// Mitsubishi GX Works2 project: project group 16 Final   PLC: FX3G

// global labels: Global1
VAR_GLOBAL
  Start_Day AT X007 : BOOL;
  Input_Oats AT D1300 : INT;
  Input_Coco AT D8100 : INT;
  Coco AT D8110 : INT;
  Oats AT D1400 : INT;
  Input_Kadaif AT D1500 : INT;
  Kadaif AT D1600 : INT;
  Input_Pistachio AT D1700 : INT;
  Pistachio AT D1800 : INT;
END_VAR
VAR_GLOBAL CONSTANT
  Zero : INT;
END_VAR
VAR_GLOBAL
  Analog_Output AT D1900 : INT;
END_VAR
VAR_GLOBAL CONSTANT
  minimum_to_start_coco : DINT := 400;  (* E_400 *)
  minimum_to_start_oats : DINT := 100;
  minimum_to_start_kadaif : DINT;
  minimum_to_start_pistachio : DINT := 60;
END_VAR
VAR_GLOBAL
  Raw_material_empty AT M2 : BOOL;
  End_Package AT M10 : BOOL;
  Work_on AT Y007 : BOOL;
  Work_Off AT M0 : BOOL;
  Start_Casting AT X003 : BOOL;
END_VAR
VAR_GLOBAL CONSTANT
  timer_casting : INT := 4;
  four_sec : INT := 40;
END_VAR
VAR_GLOBAL
  Timer_Casting_Off AT TS13 : BOOL;
  casting AT Y002 : BOOL;
  Start_Melting AT X001 : BOOL;
  Input_Chocolate AT D1100 : INT;
  HELLP AT D8140 : INT;
  Chocolate AT D1200 : INT;
END_VAR
VAR_GLOBAL CONSTANT
  minimum_to_start_Chocolate : DINT := 400;
  sub_400g : INT := 400;
END_VAR
VAR_GLOBAL
  Termo_45 AT TC9 : BOOL;
  Trmo_45 AT X002 : BOOL;
  TS2 AT TS2 : BOOL;
  Melting_Lamp AT Y001 : BOOL;
  Melting_Indicator AT X002 : BOOL;
  Sample AT X004 : BOOL;
  Save_analog_val AT D8410 : INT;
  analog_out_1 AT D8280 : INT;
END_VAR
VAR_GLOBAL CONSTANT
  Divider : INT := 400;
END_VAR
VAR_GLOBAL
  Choice AT D7000 : REAL;
END_VAR
VAR_GLOBAL CONSTANT
  Max_Oatmix : INT := 5;
  Min_Dubai : INT := 6;
END_VAR
VAR_GLOBAL
  Oat_Lamp AT M20 : BOOL;
  Dubai_Lamp AT M30 : BOOL;
  Casting_Finish AT Y002 : BOOL;
  Casting_On AT Y002 : BOOL;
END_VAR
VAR_GLOBAL CONSTANT
  Oatmix_Oat : INT := 100;
  Oatmix_Pistachio : INT := 100;
  Dubai_Oat : INT := 20;
  Dubai_Pistachio : INT := 120;
  Dubai_Kadaif : INT := 60;
END_VAR
VAR_GLOBAL
  Cannot_mix AT M40 : BOOL;
  Can_Mix AT M40 : BOOL;
  Sec5_Component AT TC5 : BOOL;
END_VAR
VAR_GLOBAL CONSTANT
  Timer_5 : INT := 50;
  timer_5_end : INT := 5;
END_VAR
VAR_GLOBAL
  Timer_End5Sec AT TS5 : BOOL;
  Flashing_Light_1 AT TC1 : BOOL;
END_VAR
VAR_GLOBAL CONSTANT
  Flashing1 : INT := 10;
END_VAR
VAR_GLOBAL
  Flashing_Light_Finish_1 AT TS1 : BOOL;
  Flashing_Lamp_1 AT Y003 : BOOL;
  Flashing_Lamp_2 AT Y004 : BOOL;
  Flashing_Light_2 AT TC2 : BOOL;
END_VAR
VAR_GLOBAL CONSTANT
  Flashing2 : INT := 10;
END_VAR
VAR_GLOBAL
  Flashing_Light_Finish_2 AT TS2 : BOOL;
  Cooling_Switch AT X006 : BOOL;
  Lamp_For_CoolingTimer AT TC12 : BOOL;
  Cooling_Lamp AT Y006 : BOOL;
  Packaging_Swich AT X000 : BOOL;
  Packaging_On AT Y005 : BOOL;
  Package_Counter AT CC3 : BOOL;
END_VAR
VAR_GLOBAL CONSTANT
  Packaging_3 : INT := 3;
END_VAR
VAR_GLOBAL
  Packaging_Counter AT CC3 : BOOL;
  Finish_Count_Packaging AT M15 : BOOL;
  Count_Packaging AT M15 : BOOL;
  Packaging_Finish AT CS3 : BOOL;
  Count_Fainal_Chocolate_Pack AT D2000 : REAL;
END_VAR
VAR_GLOBAL CONSTANT
  Constanat : INT := 1;
  Add_Pack : INT := 1;
  minimum_to_start_pistachio_100 : INT := 100;
  minimum_to_start_Chocolate_400 : INT := 400;
  minimum_to_start_oats_100 : INT := 100;
END_VAR
VAR_GLOBAL
  Material_Empty AT M2 : BOOL;
END_VAR
VAR_GLOBAL CONSTANT
  Termo_450 : INT := 450;
END_VAR
VAR_GLOBAL
  Tmer_Casting_Off AT TS1 : BOOL;
  Casting_Lamp AT M8 : BOOL;
  Pan_Count AT CC7 : BOOL;
END_VAR
VAR_GLOBAL CONSTANT
  Pan_Max : INT := 4;
END_VAR
VAR_GLOBAL
  Pan_Count_4 AT CS7 : BOOL;
  Finish_Count_Pan AT TC13 : BOOL;
  Placement_Timer AT TC8 : BOOL;
END_VAR
VAR_GLOBAL CONSTANT
  max_to_start_Chocolate_400 : INT := 400;
  minmum_to_start_oats_100 : INT := 100;
  min_to_start_Chocolate_400 : INT := 400;
  min_to_start_oats_100 : INT := 100;
  min_to_start_pistachio_100 : INT := 100;
  min_to_start_kadaif : DINT := 60;
  min_to_start_kadaif_60 : INT := 60;
END_VAR
VAR_GLOBAL
  Transfer_Coco_Lamp AT Y010 : BOOL;
END_VAR
VAR_GLOBAL CONSTANT
  Chocolate_In : INT := 400;
END_VAR
VAR_GLOBAL
  Melting_Bowl AT D2000 : INT;
END_VAR
VAR_GLOBAL CONSTANT
  Chocolate_400g : INT := 400;
END_VAR
VAR_GLOBAL
  Analog_In_1 AT D8280 : INT;
END_VAR
VAR_GLOBAL CONSTANT
  Max_Oatmix_5 : INT := 5;
  Divider_400 : INT := 400;
  Min_Dubai_6 : INT := 6;
  Min_Dubai_5 : REAL := 5;
END_VAR
VAR_GLOBAL
  Nuts AT D1400 : INT;
  Input_Nuts AT D1300 : INT;
END_VAR
VAR_GLOBAL CONSTANT
  min_to_start_nuts_100 : INT := 100;
  Max_Nuts_5 : INT := 5;
  Nutsmix_Nuts : INT := 100;
  Max_Nutsmix_5 : REAL := 5;
  Dubai_Nuts : INT := 20;
  Nuts_Mixing_Cream_200 : INT := 200;
END_VAR
VAR_GLOBAL
  Mixing_Bowl AT D2100 : INT;
END_VAR
VAR_GLOBAL CONSTANT
  Dubai_Cream_155 : INT := 155;
  Nuts_Cream_200 : INT := 200;
END_VAR
VAR_GLOBAL
  Lamp_Nuts AT M52 : BOOL;
END_VAR
VAR_GLOBAL CONSTANT
  Timer_3 : INT := 30;
END_VAR
VAR_GLOBAL
  Tempature_Reached AT X002 : BOOL;
  Melting_Indicaor_Ending AT M16 : BOOL;
  Melting_Indicator_Ending AT M16 : BOOL;
  Pan_Indicator AT X003 : BOOL;
  Pan_Located AT M45 : BOOL;
  Emergency_Swich AT X005 : BOOL;
END_VAR
VAR_GLOBAL CONSTANT
  Packaging_4 : INT := 4;
END_VAR
VAR_GLOBAL
  Timer_Cast AT TC18 : BOOL;
  Casting_Timer_4 AT TC11 : BOOL;
  Finish_Casting_Timer AT TS11 : BOOL;
  Lamp_For_CoolingTimer_Finish AT TS12 : BOOL;
  End_Of_Round AT M35 : BOOL;
  Finished_Cream AT M42 : BOOL;
END_VAR
VAR_GLOBAL CONSTANT
  Divider_10 : INT := 10;
END_VAR
VAR_GLOBAL
  AANALOG_OUTPUT AT D8282 : INT;
END_VAR
VAR_GLOBAL CONSTANT
  Multiply_40 : INT := 40;
END_VAR
VAR_GLOBAL
  storage_info AT D3020 : INT;
END_VAR
VAR_GLOBAL CONSTANT
  Multiply_400 : INT := 400;
  min_to_start_pistachio_120 : INT := 120;
  Nutmix_Pistachio : INT := 100;
END_VAR
VAR_GLOBAL
  Timer_End_5_Sec AT TS5 : BOOL;
  Sec_5_Component AT TC5 : BOOL;
  Emergency_Switch AT X005 : BOOL;
  Lamp_Cooling_Timer AT TC12 : BOOL;
  Lamp_Cooling_Timer_Finish AT TS12 : BOOL;
  Packaging_Switch AT X000 : BOOL;
  Aanalog_Output_2 AT D8282 : INT;
END_VAR

// task Task_01 (event TRUE, interval 0, priority 31): POU_01

PROGRAM POU_01
VAR CONSTANT
  Nuts_Lamp : BOOL;
END_VAR
VAR
  Timer_Casting_4 : BOOL;
  Finish_Cream : BOOL;
END_VAR
(* structured ladder/FBD written out as ST: instructions are called as NAME(EN, inputs, outputs); _pN, _eN, _tN stand for wires *)
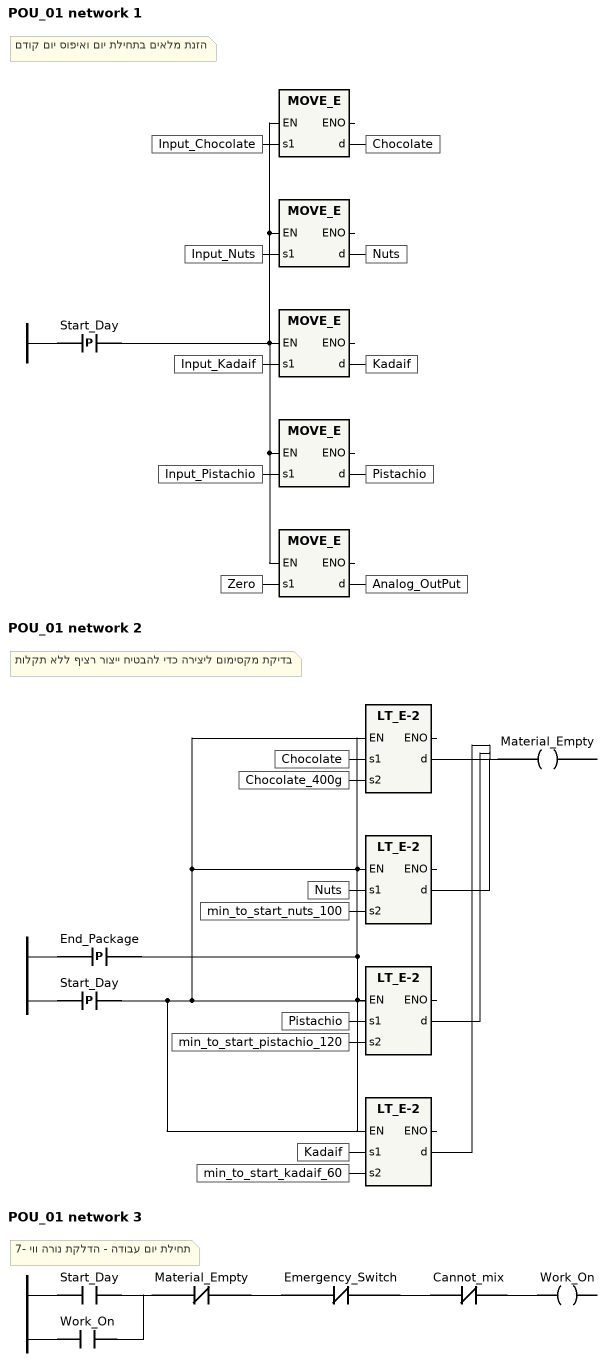
(* network 1 *)
(* הזנת מלאים בתחילת יום ואיפוס יום קודם *)
_p1 := LDP(TRUE, Start_Day);
MOVE_E(_p1, Input_Chocolate, Chocolate);
MOVE_E(_p1, Input_Nuts, Nuts);
MOVE_E(_p1, Input_Kadaif, Kadaif);
MOVE_E(_p1, Input_Pistachio, Pistachio);
MOVE_E(_p1, Zero, Analog_OutPut);
(* network 2 *)
(* בדיקת מקסימום ליצירה כדי להבטיח ייצור רציף ללא תקלות *)
_p1 := LDP(TRUE, End_Package) OR LDP(TRUE, Start_Day);
LT_E(_p1, Chocolate, Chocolate_400g, _t2);
LT_E(_p1, Nuts, min_to_start_nuts_100, _t3);
LT_E(_p1, Pistachio, min_to_start_pistachio_120, _t4);
LT_E(_p1, Kadaif, min_to_start_kadaif_60, _t5);
Material_Empty := _t2 OR _t3 OR _t4 OR _t5;
(* network 3 *)
(* תחילת יום עבודה - הדלקת נורה ווי -7 *)
Work_On := (((Start_Day OR Work_On) AND NOT Material_Empty) AND NOT Emergency_Switch) AND NOT Cannot_mix;
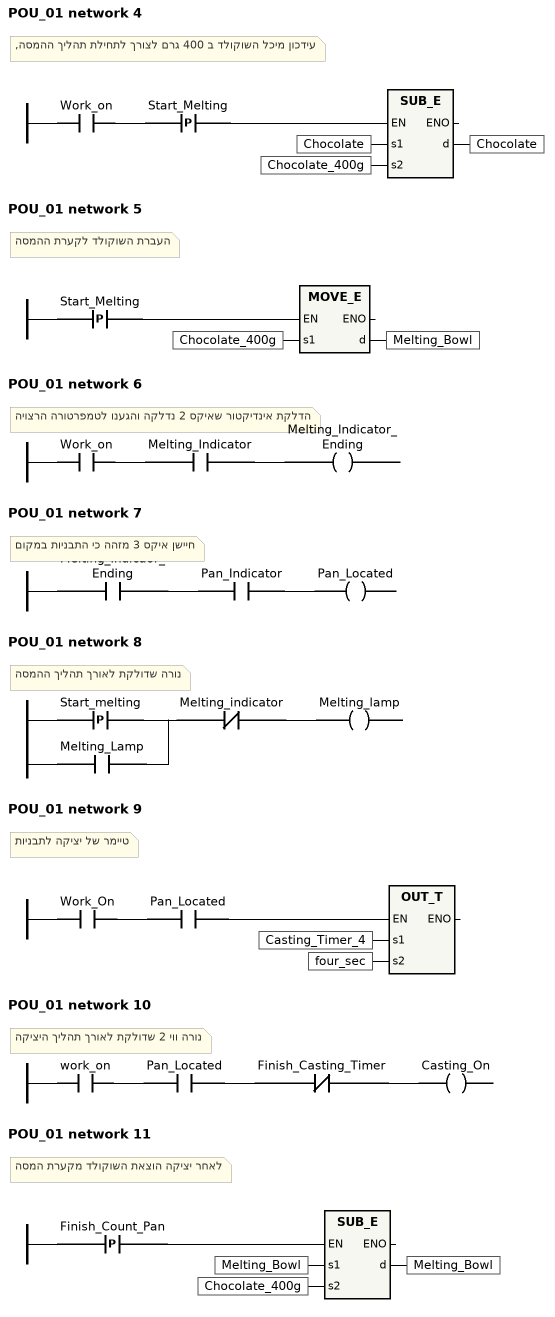
(* network 4 *)
(* עידכון מיכל השוקולד ב 400 גרם לצורך לתחילת תהליך ההמסה, *)
SUB_E(Work_on AND LDP(TRUE, Start_Melting), Chocolate, Chocolate_400g, Chocolate);
(* network 5 *)
(* העברת השוקולד לקערת ההמסה *)
MOVE_E(LDP(TRUE, Start_Melting), Chocolate_400g, Melting_Bowl);
(* network 6 *)
(* הדלקת אינדיקטור שאיקס 2 נדלקה והגענו לטמפרטורה הרצויה *)
Melting_Indicator_Ending := Work_on AND Melting_Indicator;
(* network 7 *)
(* חיישן איקס 3 מזהה כי התבניות במקום *)
Pan_Located := Melting_Indicaor_Ending AND Pan_Indicator;
(* network 8 *)
(* נורה שדולקת לאורך תהליך ההמסה *)
Melting_lamp := (LDP(TRUE, Start_melting) OR Melting_Lamp) AND NOT Melting_indicator;
(* network 9 *)
(* טיימר של יציקה לתבניות *)
OUT_T(Work_On AND Pan_Located, Casting_Timer_4, four_sec);
(* network 10 *)
(* נורה ווי 2 שדולקת לאורך תהליך היציקה *)
Casting_On := work_on AND Pan_Located AND NOT Finish_Casting_Timer;
(* network 11 *)
(* לאחר יציקה הוצאת השוקולד מקערת המסה *)
SUB_E(LDP(TRUE, Finish_Count_Pan), Melting_Bowl, Chocolate_400g, Melting_Bowl);
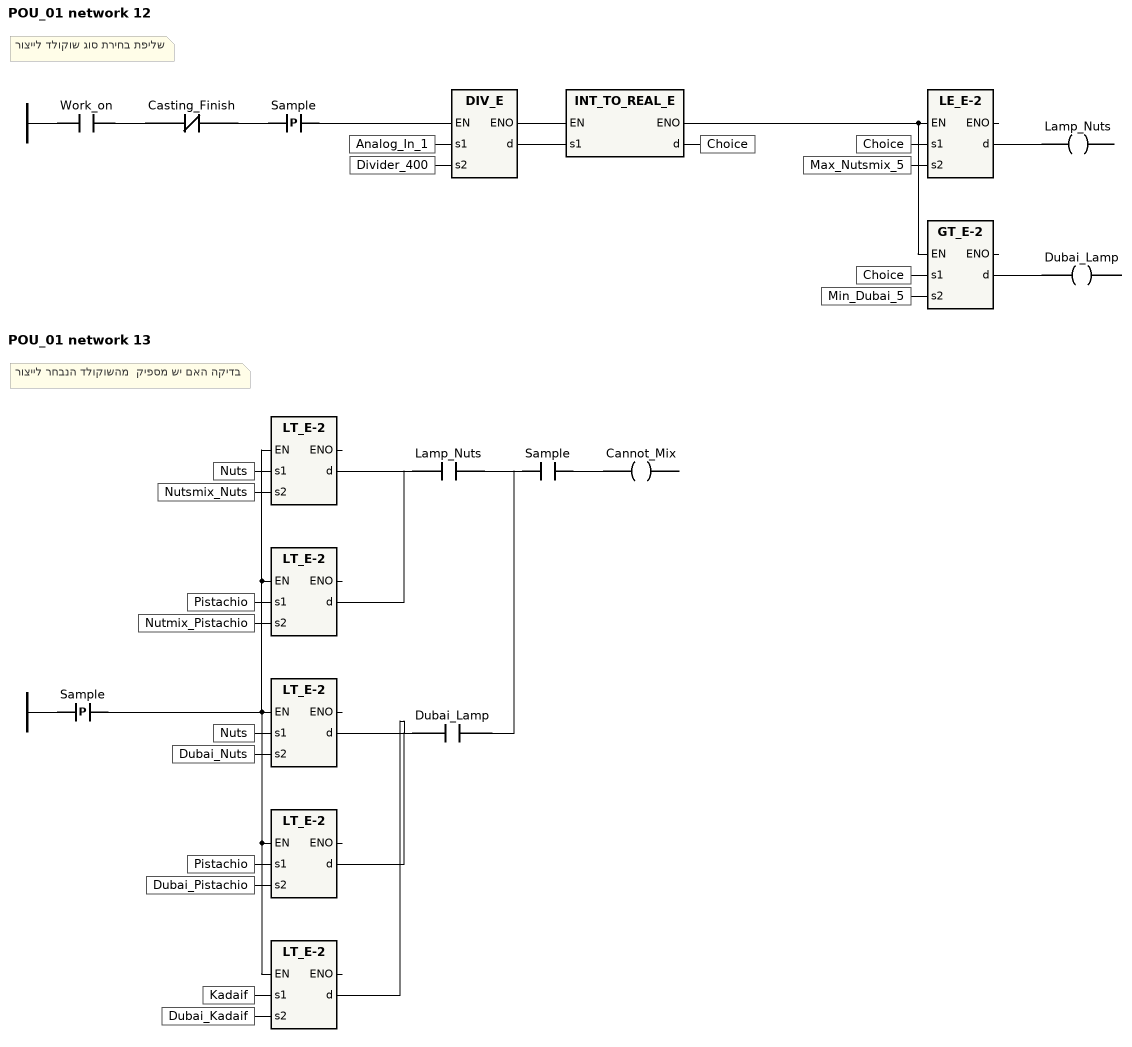
(* network 12 *)
(* שליפת בחירת סוג שוקולד לייצור *)
_e2 := DIV_E(Work_on AND NOT Casting_Finish AND LDP(TRUE, Sample), Analog_In_1, Divider_400, _t1);
_e3 := INT_TO_REAL_E(_e2, _t1, Choice);
LE_E(_e3, Choice, Max_Nutsmix_5, _t4);
Lamp_Nuts := _t4;
GT_E(_e3, Choice, Min_Dubai_5, _t5);
Dubai_Lamp := _t5;
(* network 13 *)
(* בדיקה האם יש מספיק  מהשוקולד הנבחר לייצור *)
_p1 := LDP(TRUE, Sample);
LT_E(_p1, Nuts, Nutsmix_Nuts, _t2);
LT_E(_p1, Pistachio, Nutmix_Pistachio, _t3);
LT_E(_p1, Nuts, Dubai_Nuts, _t4);
LT_E(_p1, Pistachio, Dubai_Pistachio, _t5);
LT_E(_p1, Kadaif, Dubai_Kadaif, _t6);
Cannot_Mix := (((_t2 OR _t3) AND Lamp_Nuts) OR ((_t4 OR _t5 OR _t6) AND Dubai_Lamp)) AND Sample;
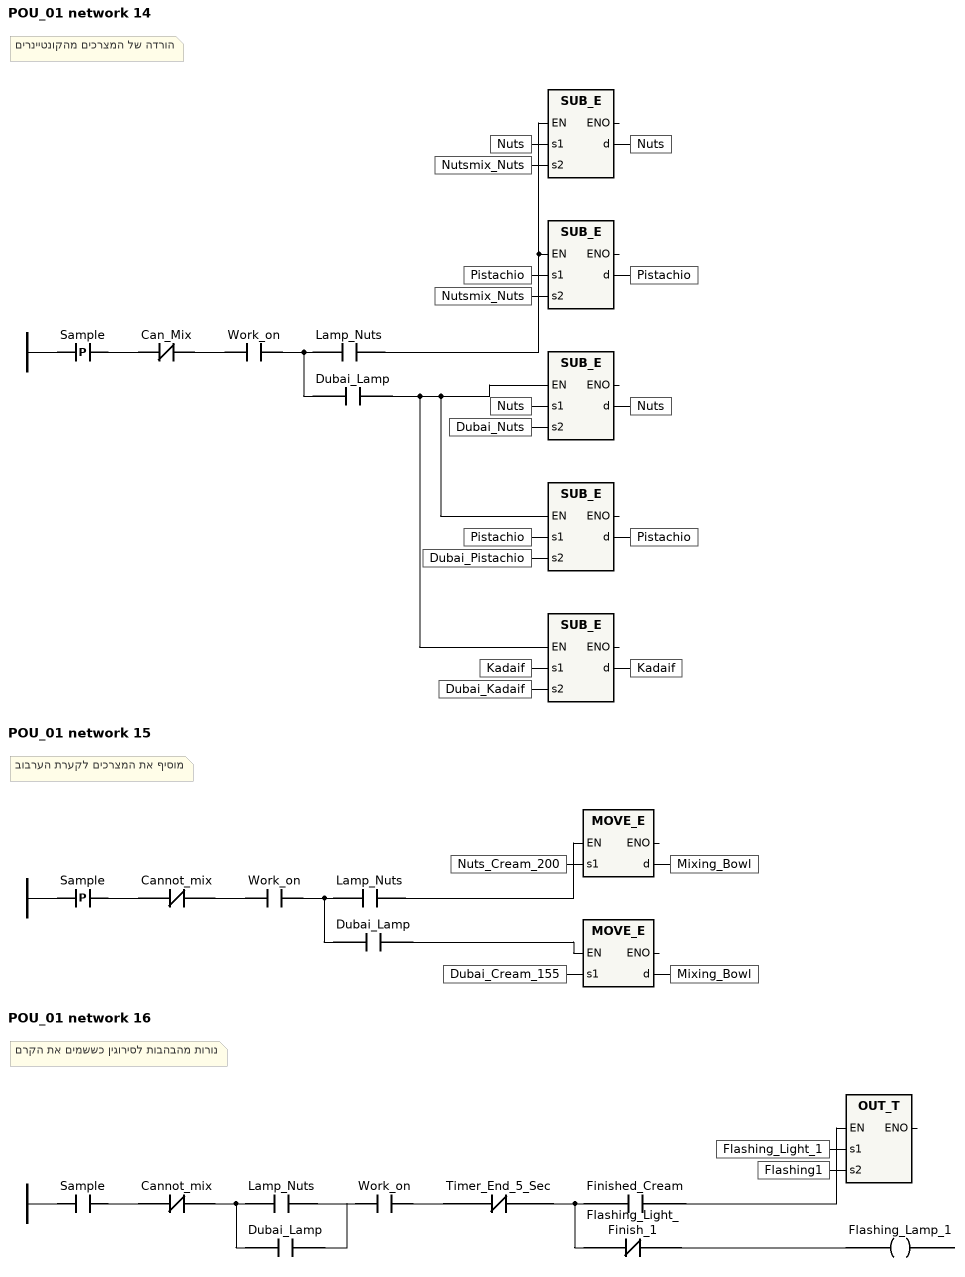
(* network 14 *)
(* הורדה של המצרכים מהקונטיינרים *)
_p1 := LDP(TRUE, Sample) AND NOT Can_Mix AND Work_on;
_p2 := _p1 AND Lamp_Nuts;
SUB_E(_p2, Nuts, Nutsmix_Nuts, Nuts);
SUB_E(_p2, Pistachio, Nutsmix_Nuts, Pistachio);
_p3 := _p1 AND Dubai_Lamp;
SUB_E(_p3, Nuts, Dubai_Nuts, Nuts);
SUB_E(_p3, Pistachio, Dubai_Pistachio, Pistachio);
SUB_E(_p3, Kadaif, Dubai_Kadaif, Kadaif);
(* network 15 *)
(* מוסיף את המצרכים לקערת הערבוב *)
_p1 := LDP(TRUE, Sample) AND NOT Cannot_mix AND Work_on;
MOVE_E(_p1 AND Lamp_Nuts, Nuts_Cream_200, Mixing_Bowl);
MOVE_E(_p1 AND Dubai_Lamp, Dubai_Cream_155, Mixing_Bowl);
(* network 16 *)
(* נורות מהבהבות לסירוגין כששמים את הקרם *)
_p1 := Sample AND NOT Cannot_mix;
_p2 := (((_p1 AND Lamp_Nuts) OR (_p1 AND Dubai_Lamp)) AND Work_on) AND NOT Timer_End_5_Sec;
OUT_T(_p2 AND Finished_Cream, Flashing_Light_1, Flashing1);
Flashing_Lamp_1 := _p2 AND NOT Flashing_Light_Finish_1;
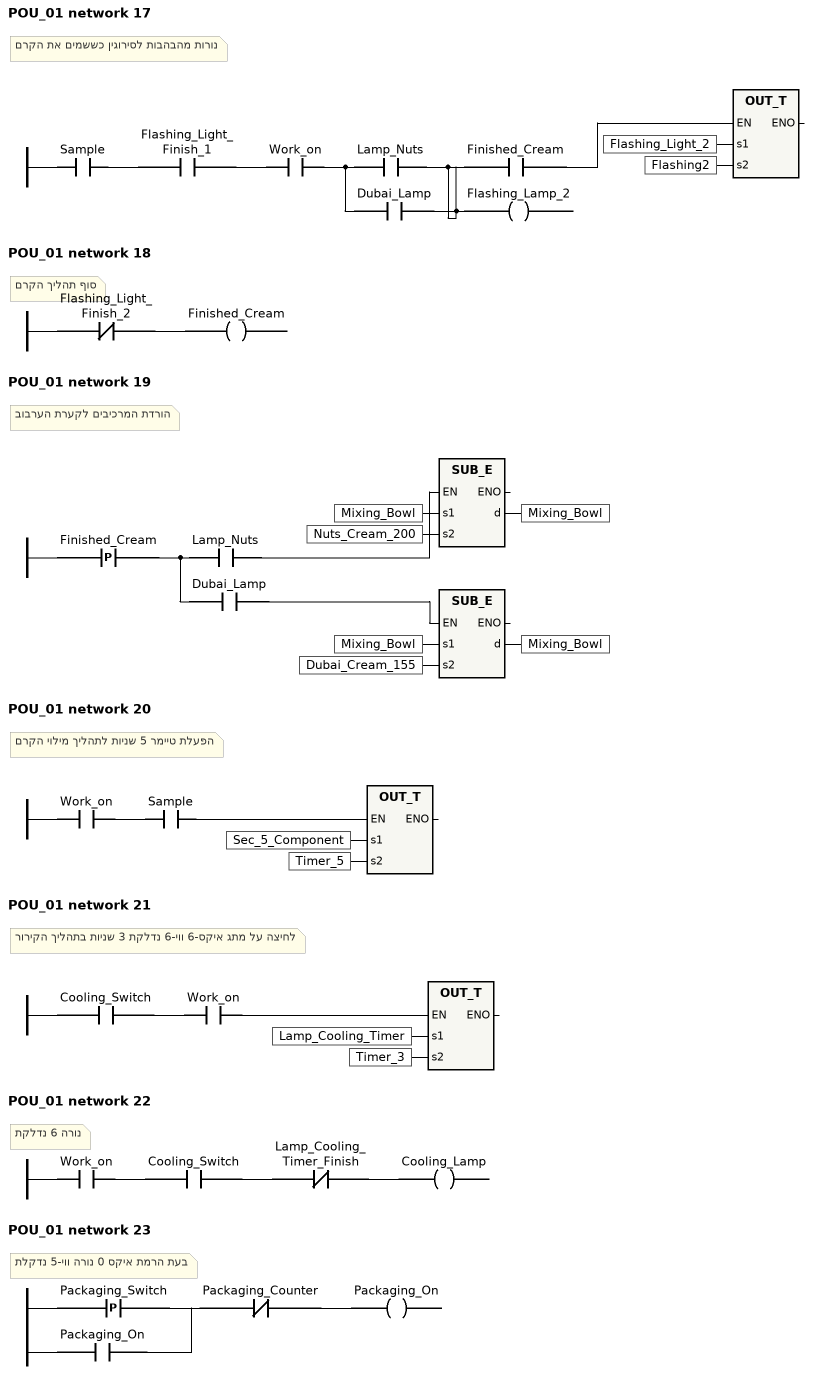
(* network 17 *)
(* נורות מהבהבות לסירוגין כששמים את הקרם *)
_p1 := Sample AND Flashing_Light_Finish_1 AND Work_on;
_p2 := (_p1 AND Lamp_Nuts) OR (_p1 AND Dubai_Lamp);
OUT_T(_p2 AND Finished_Cream, Flashing_Light_2, Flashing2);
Flashing_Lamp_2 := _p2;
(* network 18 *)
(* סוף תהליך הקרם *)
Finished_Cream := NOT Flashing_Light_Finish_2;
(* network 19 *)
(* הורדת המרכיבים לקערת הערבוב *)
_p1 := LDP(TRUE, Finished_Cream);
SUB_E(_p1 AND Lamp_Nuts, Mixing_Bowl, Nuts_Cream_200, Mixing_Bowl);
SUB_E(_p1 AND Dubai_Lamp, Mixing_Bowl, Dubai_Cream_155, Mixing_Bowl);
(* network 20 *)
(* הפעלת טיימר 5 שניות לתהליך מילוי הקרם *)
OUT_T(Work_on AND Sample, Sec_5_Component, Timer_5);
(* network 21 *)
(* לחיצה על מתג איקס-6 ווי-6 נדלקת 3 שניות בתהליך הקירור *)
OUT_T(Cooling_Switch AND Work_on, Lamp_Cooling_Timer, Timer_3);
(* network 22 *)
(* נורה 6 נדלקת *)
Cooling_Lamp := Work_on AND Cooling_Switch AND NOT Lamp_Cooling_Timer_Finish;
(* network 23 *)
(* בעת הרמת איקס 0 נורה ווי-5 נדקלת *)
Packaging_On := (LDP(TRUE, Packaging_Switch) OR Packaging_On) AND NOT Packaging_Counter;
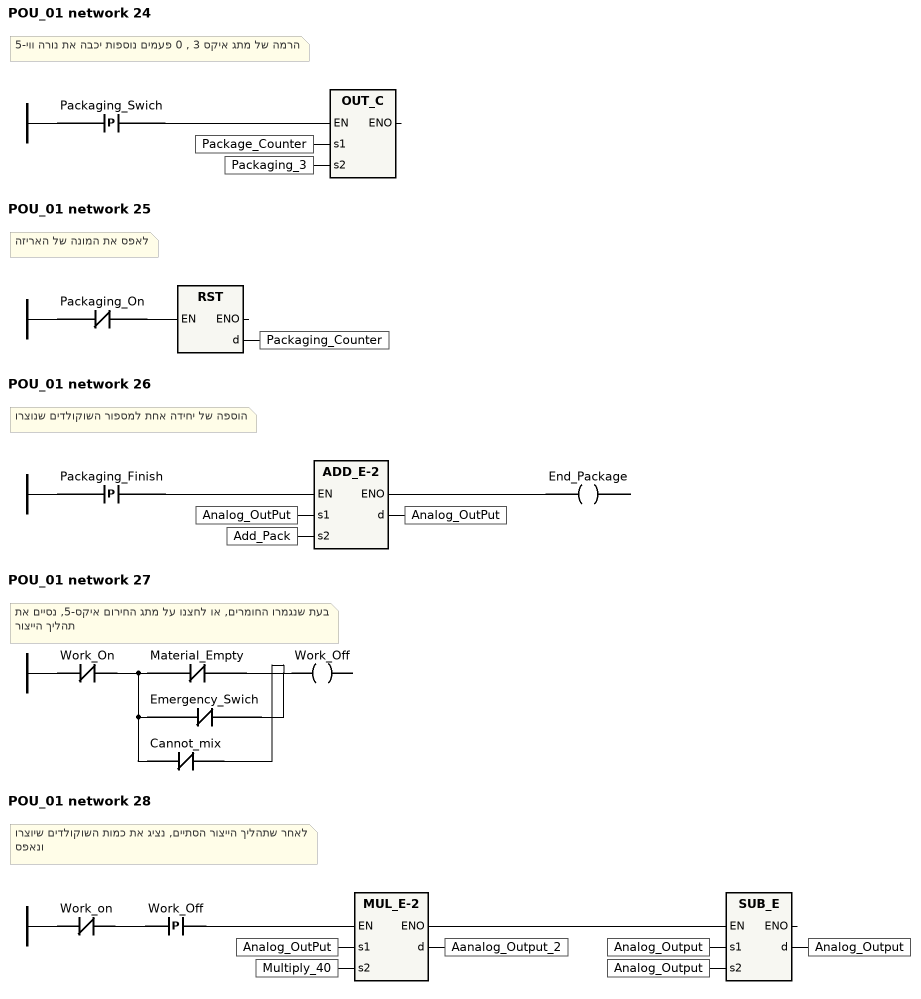
(* network 24 *)
(* הרמה של מתג איקס 0 , 3 פעמים נוספות יכבה את נורה ווי-5 *)
OUT_C(LDP(TRUE, Packaging_Swich), Package_Counter, Packaging_3);
(* network 25 *)
(* לאפס את המונה של האריזה *)
RST(NOT Packaging_On, Packaging_Counter);
(* network 26 *)
(* הוספה של יחידה אחת למספור השוקולדים שנוצרו *)
_e1 := ADD_E(LDP(TRUE, Packaging_Finish), Analog_OutPut, Add_Pack, Analog_OutPut);
End_Package := _e1;
(* network 27 *)
(* בעת שנגמרו החומרים, או לחצנו על מתג החירום איקס-5, נסיים את תהליך הייצור *)
_p1 := NOT Work_On;
Work_Off := (_p1 AND NOT Material_Empty) OR (_p1 AND NOT Emergency_Swich) OR (_p1 AND NOT Cannot_mix);
(* network 28 *)
(* לאחר שתהליך הייצור הסתיים, נציג את כמות השוקולדים שיוצרו ונאפס *)
_e1 := MUL_E(NOT Work_on AND LDP(TRUE, Work_Off), Analog_OutPut, Multiply_40, Aanalog_Output_2);
SUB_E(_e1, Analog_Output, Analog_Output, Analog_Output);
END_PROGRAM
